TYPE ConveyorConfiguration :
STRUCT
	iNumSensor : DINT;
	iNumRamp : DINT;
	iNumPusher : DINT;
END_STRUCT
END_TYPE

(* stored: Version 1.1.0.1
   DUT ConveyorConfiguration: Id {c45f872a-c89f-4045-be49-aabd68bcc7a6} *)
